TYPE LaserConfigs :
STRUCT
	SMD12LaserConfig : SMD12LaserConfig;
	Piano450LaserConfig : Piano450LaserConfig;
	Sapphire488LaserConfig : Sapphire488LaserConfig;
END_STRUCT
END_TYPE

(* stored: Version 1.1.0.1, ProductVersion 3.1.4024.12
   DUT LaserConfigs: Id {df745186-20cc-409d-b80d-67bb6928cd30} *)
